Fanuc TP program (LS listing): AWFILL.LS

/PROG  AWFILL
/ATTR
OWNER		= MNEDITOR;
COMMENT		= "AwFill";
PROG_SIZE	= 0;
CREATE		= DATE 26-01-01  TIME 00:00:00;
MODIFIED	= DATE 26-01-01  TIME 00:00:00;
FILE_NAME	= ;
VERSION		= 0;
LINE_COUNT	= 11;
MEMORY_SIZE	= 0;
PROTECT		= READ_WRITE;
TCD:  STACK_SIZE	= 0,
      TASK_PRIORITY	= 50,
      TIME_SLICE	= 0,
      BUSY_LAMP_OFF	= 0,
      ABORT_REQUEST	= 0,
      PAUSE_REQUEST	= 0;
DEFAULT_GROUP	= 1,*,*,*,*;
CONTROL_CODE	= 00000000 00000000;
/MN
   1:  !RAPID ArrayWriteProbe.AwFill ;
   2:  FOR R[1:i]=1 TO 3 ;
   3:  FOR R[2:j]=1 TO 4 ;
   4:  R[3:NumberIndex]=R[1:i]    ;
   5:  R[3:NumberIndex]=R[3:NumberIndex]*4    ;
   6:  R[3:NumberIndex]=R[3:NumberIndex]+R[2:j]    ;
   7:  R[3:NumberIndex]=R[3:NumberIndex]+184    ;
   8:  R[4:Calc1]=R[1:i]*10    ;
   9:  R[R[3]]=R[4:Calc1]+R[2:j]    ;
  10:  ENDFOR ;
  11:  ENDFOR ;
/POS
/END
